(* PLC project flour, Dassault Systèmes ControlBuild 2024x *)
(* stored: creationDateTime 2023-10-03T11:13:38-01:00 *)

FUNCTION_BLOCK faults
  VAR_INPUT
    generalFault3 : BOOL := false;
    generalFault2 : BOOL := false;
    generalFault1 : BOOL := false;
  END_VAR
  VAR_OUTPUT
    fault : BOOL := false;
  END_VAR

(* LD diagram, written out as Structured Text *)
1:
fault := generalFault3 OR generalFault1 OR generalFault2;
END_FUNCTION_BLOCK

PROGRAM batch.flour
  VAR_INPUT
    cycleInProgress : BOOL := false;
    acknowledgePB : BOOL := false;
    weighingRequest : BOOL := false;
  END_VAR
  VAR_INPUT
    flourWeight : DINT := 0;
  END_VAR
  VAR_INPUT
    autoMode : BOOL := false;
    manualMode : BOOL := false;
  END_VAR
  VAR_OUTPUT
    flourExtraction : REAL := 0.0;
    weighingOk : BOOL := false;
    fault : BOOL := false;
  END_VAR

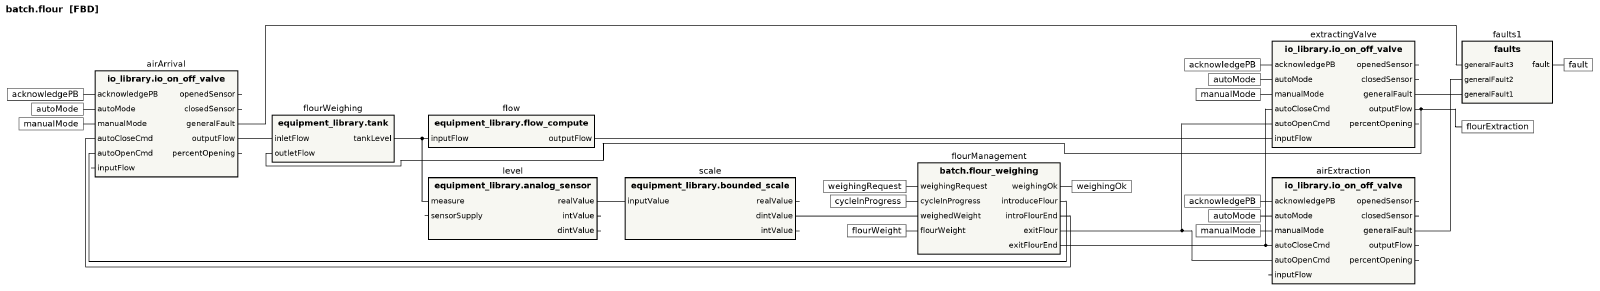
(* FBD diagram, written out as Structured Text *)
airArrival(acknowledgePB := acknowledgePB, autoMode := autoMode, manualMode := manualMode, autoCloseCmd := flourManagement.introFlourEnd, autoOpenCmd := flourManagement.introduceFlour);
flow(inputFlow := flourWeighing.tankLevel);
extractingValve(acknowledgePB := acknowledgePB, autoMode := autoMode, manualMode := manualMode, autoCloseCmd := flourManagement.exitFlourEnd, autoOpenCmd := flourManagement.exitFlour, inputFlow := flow.outputFlow);
flourWeighing(inletFlow := airArrival.outputFlow, outletFlow := extractingValve.outputFlow);
level(measure := flourWeighing.tankLevel);
scale(inputValue := level.realValue);
flourManagement(weighingRequest := weighingRequest, cycleInProgress := cycleInProgress, weighedWeight := scale.dintValue, flourWeight := flourWeight);
weighingOk := flourManagement.weighingOk;
airExtraction(acknowledgePB := acknowledgePB, autoMode := autoMode, manualMode := manualMode, autoCloseCmd := flourManagement.exitFlourEnd, autoOpenCmd := flourManagement.exitFlour);
faults1(generalFault3 := airArrival.generalFault, generalFault2 := airExtraction.generalFault, generalFault1 := extractingValve.generalFault);
fault := faults1.fault;
flourExtraction := extractingValve.outputFlow;
END_PROGRAM
